// ---- 20_Product/20_ProBox/40_TC_Visualization/14_Group/V_Group.TcVIS
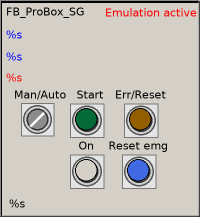
VISUALIZATION V_Group  // 200x217
VAR_IN_OUT
	{attribute 'VAR_IN_OUT_AS_POINTER'}
	fbFunction		: FB_ProBOXSG;
	fbEmuFunction	: FB_ProBOXSG_Emulation;
END_VAR
    Rectangle (0,1 200x216)
    Rectangle (6,194 177x20), "%s", text variable: fbFunction.ConfigGroup.GroupName
    Label (3,2 158x20), "FB_ProBox_SG"
    Rectangle (3,25 99x20), "%s", text variable: fbFunction.GroupData.OperationState.eState
    Rectangle (3,68 161x20), "%s", tooltip "%s", text variable: fbFunction.GroupData.ErrorData.Error.ErrorCode.Conv, invisible if: fbFunction.GroupData.ErrorData.Error.ErrorCode.Conv = 0
        p4168582468: fbFunction.GroupData.ErrorData.Error.ErrorParam
    Rectangle (3,47 99x20), "%s", text variable: fbFunction.GroupData.OperationState.eMode
    RotarySwitch (21,103 33x33), variable: fbEmuFunction.DebugManualModeSw, behaviour: TOGGLE, style: Switch-RotarySwitch-Gray
    Label (11,84 58x22), "Man/Auto"
    Rectangle (102,3 95x20), "Emulation active", invisible if: NOT ProBoxSystem.EMULATION_ENABLED
    PushSwitch (70,103 34x35), behaviour: TOGGLE, style: Switch-PushSwitch-Gray
    Ellipse (75,108 22x22), colour toggle: fbFunction.HW_Outputs.GroupStarted
        tap fbEmuFunction.DebugStartButton
    Label (71,84 38x22), "Start"
    Label (106,84 69x22), "Err/Reset"
    PushSwitch (124,103 34x35), behaviour: TOGGLE, style: Switch-PushSwitch-Gray
    Ellipse (129,108 22x22), colour toggle: fbFunction.HW_Outputs.ErrorPending
        tap fbEmuFunction.DebugResetButton
    Label (52,135 69x22), "On"
    PushSwitch (70,154 34x35), behaviour: TOGGLE, style: Switch-PushSwitch-Gray
    Ellipse (75,159 22x22), colour toggle: fbFunction.HW_Outputs.MainContactorLamp
        tap fbEmuFunction.DebugMcOnButton
    PushSwitch (122,154 34x35), behaviour: TOGGLE, style: Switch-PushSwitch-Gray
    Ellipse (127,159 22x22), colour toggle: fbFunction.HW_Outputs.EmergencyLamp
        tap fbEmuFunction.DebugResetEmgButton
    Label (104,135 69x22), "Reset emg"
END_VISUALIZATION

// ---- 20_Product/20_ProBox/40_TC_Visualization/15_PowerStore/AccessPanelCmbTxtList.TcTLO
TEXTLIST AccessPanelCmbTxtList
  1 = '1'
  2 = '2'
  3 = '3'
  4 = '4'
   = ''
END_TEXTLIST

// ---- 20_Product/20_ProBox/40_TC_Visualization/15_PowerStore/AkCmbTxtList.TcTLO
TEXTLIST AkCmbTxtList
  1 = '1'
  2 = '2'
  3 = '3'
  4 = '4'
   = ''
END_TEXTLIST

// ---- 20_Product/20_ProBox/40_TC_Visualization/15_PowerStore/LevelCmbTxtList.TcTLO
TEXTLIST LevelCmbTxtList
  1 = '1'
  2 = '2'
  3 = '3'
  4 = '4'
  5 = '5'
  6 = '6'
  7 = '7'
  8 = '8'
  9 = '9'
  10 = '10'
  11 = '11'
  12 = '12'
   = ''
END_TEXTLIST

// ---- 20_Product/20_ProBox/40_TC_Visualization/15_PowerStore/PanelCmbTxtList.TcTLO
TEXTLIST PanelCmbTxtList
  1 = '1'
  2 = '2'
  3 = '3'
  4 = '4'
   = ''
END_TEXTLIST

// ---- 20_Product/20_ProBox/40_TC_Visualization/15_PowerStore/TransferPanelCmbTxtList.TcTLO
TEXTLIST TransferPanelCmbTxtList
  1 = '1'
  2 = '2'
  3 = '3'
  4 = '4'
   = ''
END_TEXTLIST

// ---- 20_Product/20_ProBox/40_TC_Visualization/15_PowerStore/V_AccessPanel.TcVIS
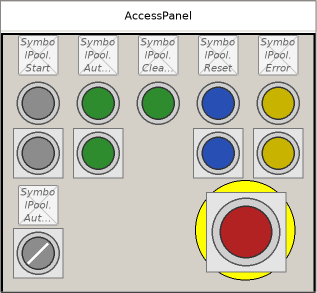
VISUALIZATION V_AccessPanel  // 317x293
VAR_IN_OUT
	Signals  : ST_AccessPanel;
END_VAR
    Rectangle (1,33 314x260)
    Image (18,35 40x40), image: SymbolPool.Start
    PushSwitch (13,128 50x50), tooltip "Activate main contactor", variable: Signals.inputs.PB_ActivateMainContactor, behaviour: TAP, style: Switch-PushSwitch-Gray
    Lamp1 (13,78 50x50), tooltip "Main contactor activated", variable: Signals.outputs.LED_MainContactorActivated, style: Lamp-Lamp1-Gray
    PushSwitch (73,128 50x50), tooltip "Auto on", variable: Signals.inputs.PB_AutoOn, behaviour: TAP, style: Switch-PushSwitch-Green
    Lamp1 (73,78 50x50), tooltip "Auto activated", variable: Signals.outputs.LED_AutoIsOn, style: Lamp-Lamp1-Green
    Lamp1 (133,78 50x50), tooltip "Clear enterance", variable: Signals.outputs.LED_ClearEnterance, style: Lamp-Lamp1-Green
    Lamp1 (193,78 50x50), tooltip "Emergency stop", variable: Signals.outputs.LED_EmergencyStop, style: Lamp-Lamp1-Blue
    PushSwitch (193,128 50x50), tooltip "Reset emergency stop", variable: Signals.inputs.PB_EmergencyStopReset, behaviour: TAP, style: Switch-PushSwitch-Blue
    Lamp1 (253,78 50x50), tooltip "Error", variable: Signals.outputs.LED_Error, style: Lamp-Lamp1-Yellow
    PushSwitch (253,128 50x50), tooltip "Reset error", variable: Signals.inputs.PB_ErrorReset, behaviour: TAP, style: Switch-PushSwitch-Yellow
    RotarySwitch (13,228 50x50), tooltip "Auto/Entry request key switch", variable: Signals.inputs.SW_EntryRequest, behaviour: TOGGLE, style: Switch-RotarySwitch-Gray
    Ellipse (195,180 100x100)
    PushSwitch (206,192 80x80), variable: Signals.inputs.PB_EmergencyStop, behaviour: TOGGLE, style: Switch-PushSwitch-Red
    Image (78,35 40x40), image: SymbolPool.AutoOn
    Image (138,35 40x40), image: SymbolPool.ClearToEnter
    Image (198,35 40x40), image: SymbolPool.Reset
    Image (258,35 40x40), image: SymbolPool.Error
    Image (18,185 40x40), image: SymbolPool.AutoMan
    Textfield (0,1 317x30), "AccessPanel"
END_VISUALIZATION

// ---- 20_Product/20_ProBox/40_TC_Visualization/15_PowerStore/V_AKcabinetPanel.TcVIS
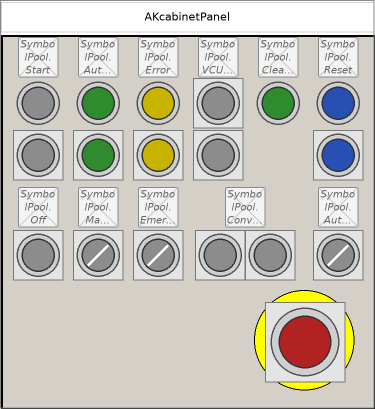
VISUALIZATION V_AKcabinetPanel  // 375x409
VAR_IN_OUT
	Signals : ST_AKcabinetPanel;
END_VAR
    Rectangle (1,35 374x374)
    Lamp1 (13,78 50x50), tooltip "Main contactor activeated", variable: Signals.outputs.LED_MainContactorActivated, style: Lamp-Lamp1-Gray
    PushSwitch (13,130 50x50), tooltip "Activate main contactor", variable: Signals.inputs.PB_ActivateMainContactor, behaviour: TAP, style: Switch-PushSwitch-Gray
    PushSwitch (73,130 50x50), tooltip "Auto on", variable: Signals.inputs.PB_AutoOn, behaviour: TAP, style: Switch-PushSwitch-Green
    Lamp1 (73,78 50x50), tooltip "Auto activated", variable: Signals.outputs.LED_AutoIsOn, style: Lamp-Lamp1-Green
    Lamp1 (133,78 50x50), tooltip "Error", variable: Signals.outputs.LED_Error, style: Lamp-Lamp1-Yellow
    PushSwitch (133,130 50x50), tooltip "Reset error", variable: Signals.inputs.PB_ErrorReset, behaviour: TAP, style: Switch-PushSwitch-Yellow
    RotarySwitch (73,230 50x50), tooltip "Man/Auto key switch", variable: Signals.inputs.SW_Auto, behaviour: TOGGLE, style: Switch-RotarySwitch-Gray
    PushSwitch (13,230 50x50), tooltip "Main contactor off", variable: Signals.inputs.PB_MainContactorOff, behaviour: TAP, style: Switch-PushSwitch-Gray
    Image (18,37 40x40), image: SymbolPool.Start
    Image (78,37 40x40), image: SymbolPool.AutoOn
    Image (138,37 40x40), image: SymbolPool.Error
    Image (18,187 40x40), image: SymbolPool.Off
    Image (78,187 40x40), image: SymbolPool.ManAuto
    Image (198,37 40x40), image: SymbolPool.VCUpDown
    PushSwitch (193,130 50x50), tooltip "VC Down", variable: Signals.inputs.PB_VcDown, behaviour: TAP, style: Switch-PushSwitch-Gray
    PushSwitch (193,78 50x50), tooltip "VC Up", variable: Signals.inputs.PB_VcUp, behaviour: TAP, style: Switch-PushSwitch-Gray
    Lamp1 (253,78 50x50), tooltip "Clear enterance", variable: Signals.outputs.LED_ClearEnterance, style: Lamp-Lamp1-Green
    Lamp1 (313,78 50x50), tooltip "Emergency stop", variable: Signals.outputs.LED_EmergencyStop, style: Lamp-Lamp1-Blue
    PushSwitch (313,130 50x50), tooltip "Reset emergency stop", variable: Signals.inputs.PB_EmergencyStopReset, behaviour: TAP, style: Switch-PushSwitch-Blue
    Image (258,37 40x40), image: SymbolPool.ClearToEnter
    Image (318,37 40x40), image: SymbolPool.Reset
    Image (225,187 40x40), image: SymbolPool.Conv_L_R
    PushSwitch (245,230 50x50), tooltip "VC Conveyor Right", variable: Signals.inputs.PB_VcConvRight, behaviour: TAP, style: Switch-PushSwitch-Gray
    PushSwitch (195,230 50x50), tooltip "VC Conveyor Left", variable: Signals.inputs.PB_VcConvLeft, behaviour: TAP, style: Switch-PushSwitch-Gray
    Image (318,187 40x40), image: SymbolPool.AutoMan
    RotarySwitch (313,230 50x50), tooltip "Auto/Entry request key switch", variable: Signals.inputs.SW_EntryRequest, behaviour: TOGGLE, style: Switch-RotarySwitch-Gray
    RotarySwitch (133,230 50x50), tooltip "Emergency drive key switch", variable: Signals.inputs.SW_EmergencyDrive, behaviour: TOGGLE, style: Switch-RotarySwitch-Gray
    Image (138,187 40x40), image: SymbolPool.EmergencyDrive
    Ellipse (254,290 100x100)
    PushSwitch (265,302 80x80), variable: Signals.inputs.PB_EmergencyStop, behaviour: TOGGLE, style: Switch-PushSwitch-Red
    Textfield (1,2 373x30), "AKcabinetPanel"
END_VISUALIZATION

// ---- 20_Product/20_ProBox/40_TC_Visualization/15_PowerStore/V_AkPanelSelecCmb.TcVIS
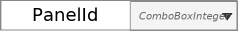
VISUALIZATION V_AkPanelSelecCmb  // 238x31
    ComboBoxInteger (130,1 108x30), variable: VisuGVL.fbPanelImp.AKPanelId, text list: 'AkCmbTxtList'
    Textfield (1,0 129x30), "PanelId"
END_VISUALIZATION

// ---- 20_Product/20_ProBox/40_TC_Visualization/15_PowerStore/V_ApSelecCmb.TcVIS
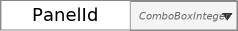
VISUALIZATION V_ApSelecCmb  // 238x31
    ComboBoxInteger (130,1 108x30), variable: VisuGVL.fbPanelImp.PanelId, text list: 'PanelCmbTxtList'
    Textfield (1,0 129x30), "PanelId"
END_VISUALIZATION

// ---- 20_Product/20_ProBox/40_TC_Visualization/15_PowerStore/V_LevelSelecCmb.TcVIS
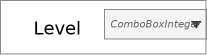
VISUALIZATION V_LevelSelecCmb  // 207x55
    ComboBoxInteger (104,9 103x30), variable: VisuGVL.fbPanelImp.Level, text list: 'LevelCmbTxtList'
    Label (5,2 105x53), "Level"
END_VISUALIZATION

// ---- 20_Product/20_ProBox/40_TC_Visualization/15_PowerStore/V_PanelSelecCmb.TcVIS
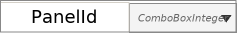
VISUALIZATION V_PanelSelecCmb  // 237x33
    ComboBoxInteger (129,3 108x30), variable: VisuGVL.fbPanelImp.PanelId, text list: 'PanelCmbTxtList'
    Textfield (0,2 129x30), "PanelId"
END_VISUALIZATION

// ---- 20_Product/20_ProBox/40_TC_Visualization/15_PowerStore/V_TpSelecCmb.TcVIS
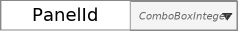
VISUALIZATION V_TpSelecCmb  // 238x31
    ComboBoxInteger (130,1 108x30), variable: VisuGVL.fbPanelImp.PanelId, text list: 'PanelCmbTxtList'
    Textfield (1,0 129x30), "PanelId"
END_VISUALIZATION

// ---- 20_Product/20_ProBox/40_TC_Visualization/15_PowerStore/V_TransferPanel.TcVIS
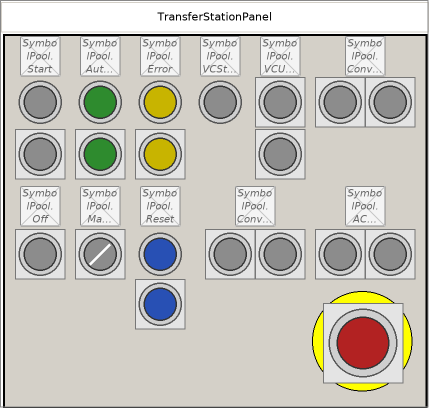
VISUALIZATION V_TransferPanel  // 429x408
VAR_IN_OUT
	Signals : ST_TransferPanel;
END_VAR
    Rectangle (3,34 424x374)
    Ellipse (312,291 100x100)
    PushSwitch (15,129 50x50), tooltip "Activate main contactor", variable: Signals.inputs.PB_ActivateMainContactor, behaviour: TAP, style: Switch-PushSwitch-Gray
    Lamp1 (15,77 50x50), tooltip "Main contactor activeated", variable: Signals.outputs.LED_MainContactorActivated, style: Lamp-Lamp1-Gray
    PushSwitch (75,129 50x50), tooltip "Auto on", variable: Signals.inputs.PB_AutoOn, behaviour: TAP, style: Switch-PushSwitch-Green
    Lamp1 (75,77 50x50), tooltip "Auto activated", variable: Signals.outputs.LED_AutoIsOn, style: Lamp-Lamp1-Green
    Lamp1 (135,77 50x50), tooltip "Error", variable: Signals.outputs.LED_Error, style: Lamp-Lamp1-Yellow
    PushSwitch (135,129 50x50), tooltip "Reset error", variable: Signals.inputs.PB_ErrorReset, behaviour: TAP, style: Switch-PushSwitch-Yellow
    Lamp1 (135,229 50x50), tooltip "Emergency stop", variable: Signals.outputs.LED_EmergencyStop, style: Lamp-Lamp1-Blue
    PushSwitch (135,279 50x50), tooltip "Reset emergency stop", variable: Signals.inputs.PB_EmergencyStopReset, behaviour: TAP, style: Switch-PushSwitch-Blue
    RotarySwitch (75,229 50x50), tooltip "Man/Auto", variable: Signals.inputs.SW_Auto, behaviour: TOGGLE, style: Switch-RotarySwitch-Gray
    Lamp1 (195,77 50x50), tooltip "VC stopped", variable: Signals.outputs.LED_VcStopped, style: Lamp-Lamp1-Gray
    PushSwitch (255,129 50x50), tooltip "VC Down", variable: Signals.inputs.PB_VcDown, behaviour: TAP, style: Switch-PushSwitch-Gray
    PushSwitch (255,77 50x50), tooltip "VC Up", variable: Signals.inputs.PB_VcUp, behaviour: TAP, style: Switch-PushSwitch-Gray
    PushSwitch (365,77 50x50), tooltip "Transfer Conveyor Right", variable: Signals.inputs.PB_Conv_1_Right, behaviour: TAP, style: Switch-PushSwitch-Gray
    PushSwitch (315,77 50x50), tooltip "Transfer Conveyor Left", variable: Signals.inputs.PB_Conv_1_Left, behaviour: TAP, style: Switch-PushSwitch-Gray
    PushSwitch (255,229 50x50), tooltip "VC Conveyor Right", variable: Signals.inputs.PB_VcConvRight, behaviour: TAP, style: Switch-PushSwitch-Gray
    PushSwitch (205,229 50x50), tooltip "VC Conveyor Left", variable: Signals.inputs.PB_VcConvLeft, behaviour: TAP, style: Switch-PushSwitch-Gray
    PushSwitch (365,229 50x50), tooltip "AC Conveyor Right", variable: Signals.inputs.PB_AC_ConvRight, behaviour: TAP, style: Switch-PushSwitch-Gray
    PushSwitch (315,229 50x50), tooltip "AC Conveyor Left", variable: Signals.inputs.PB_AC_ConvLeft, behaviour: TAP, style: Switch-PushSwitch-Gray
    PushSwitch (15,229 50x50), tooltip "Main contactor off", variable: Signals.inputs.PB_MainContactorOff, behaviour: TAP, style: Switch-PushSwitch-Gray
    PushSwitch (323,303 80x80), tooltip "Emergency stop", variable: Signals.inputs.PB_EmergencyStop, behaviour: TOGGLE, style: Switch-PushSwitch-Red
    Image (20,36 40x40), image: SymbolPool.Start
    Image (80,36 40x40), image: SymbolPool.AutoOn
    Image (140,36 40x40), image: SymbolPool.Error
    Image (200,36 40x40), image: SymbolPool.VCStopped
    Image (260,36 40x40), image: SymbolPool.VCUpDown
    Image (345,36 40x40), image: SymbolPool.Conv1_L_R
    Image (235,186 40x40), image: SymbolPool.Conv_L_R
    Image (345,186 40x40), image: SymbolPool.AC_Conv_L_R
    Image (20,186 40x40), image: SymbolPool.Off
    Image (80,186 40x40), image: SymbolPool.ManAuto
    Image (140,186 40x40), image: SymbolPool.Reset
    Textfield (1,2 428x30), "TransferStationPanel"
END_VISUALIZATION

// ---- 20_Product/20_ProBox/40_TC_Visualization/15_PowerStore/V_VC_AccessPanel.TcVIS
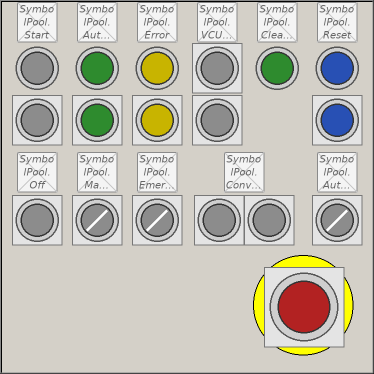
VISUALIZATION V_VC_AccessPanel  // 374x374
VAR_IN_OUT
	Signals : ST_VC_AccessPanel;
END_VAR
    Rectangle (0,0 374x374)
    Lamp1 (12,43 50x50), tooltip "Main contactor activeated", variable: Signals.outputs.LED_MainContactorActivated, style: Lamp-Lamp1-Gray
    PushSwitch (12,95 50x50), tooltip "Activate main contactor", variable: Signals.inputs.PB_ActivateMainContactor, behaviour: TAP, style: Switch-PushSwitch-Gray
    PushSwitch (72,95 50x50), tooltip "Auto on", variable: Signals.inputs.PB_AutoOn, behaviour: TAP, style: Switch-PushSwitch-Green
    Lamp1 (72,43 50x50), tooltip "Auto activated", variable: Signals.outputs.LED_AutoIsOn, style: Lamp-Lamp1-Green
    Lamp1 (132,43 50x50), tooltip "Error", variable: Signals.outputs.LED_Error, style: Lamp-Lamp1-Yellow
    PushSwitch (132,95 50x50), tooltip "Reset error", variable: Signals.inputs.PB_ErrorReset, behaviour: TAP, style: Switch-PushSwitch-Yellow
    RotarySwitch (72,195 50x50), tooltip "Man/Auto key switch", variable: Signals.inputs.SW_Auto, behaviour: TOGGLE, style: Switch-RotarySwitch-Gray
    PushSwitch (12,195 50x50), tooltip "Main contactor off", variable: Signals.inputs.PB_MainContactorOff, behaviour: TAP, style: Switch-PushSwitch-Gray
    Image (17,2 40x40), image: SymbolPool.Start
    Image (77,2 40x40), image: SymbolPool.AutoOn
    Image (137,2 40x40), image: SymbolPool.Error
    Image (17,152 40x40), image: SymbolPool.Off
    Image (77,152 40x40), image: SymbolPool.ManAuto
    Image (197,2 40x40), image: SymbolPool.VCUpDown
    PushSwitch (192,95 50x50), tooltip "VC Down", variable: Signals.inputs.PB_VcDown, behaviour: TAP, style: Switch-PushSwitch-Gray
    PushSwitch (192,43 50x50), tooltip "VC Up", variable: Signals.inputs.PB_VcUp, behaviour: TAP, style: Switch-PushSwitch-Gray
    Lamp1 (252,43 50x50), tooltip "Clear enterance", variable: Signals.outputs.LED_ClearEnterance, style: Lamp-Lamp1-Green
    Lamp1 (312,43 50x50), tooltip "Emergency stop", variable: Signals.outputs.LED_EmergencyStop, style: Lamp-Lamp1-Blue
    PushSwitch (312,95 50x50), tooltip "Reset emergency stop", variable: Signals.inputs.PB_EmergencyStopReset, behaviour: TAP, style: Switch-PushSwitch-Blue
    Image (257,2 40x40), image: SymbolPool.ClearToEnter
    Image (317,2 40x40), image: SymbolPool.Reset
    Image (224,152 40x40), image: SymbolPool.Conv_L_R
    PushSwitch (244,195 50x50), tooltip "VC Conveyor Right", variable: Signals.inputs.PB_VcConvRight, behaviour: TAP, style: Switch-PushSwitch-Gray
    PushSwitch (194,195 50x50), tooltip "VC Conveyor Left", variable: Signals.inputs.PB_VcConvLeft, behaviour: TAP, style: Switch-PushSwitch-Gray
    Image (317,152 40x40), image: SymbolPool.AutoMan
    RotarySwitch (312,195 50x50), tooltip "Auto/Entry request key switch", variable: Signals.inputs.SW_EntryRequest, behaviour: TOGGLE, style: Switch-RotarySwitch-Gray
    RotarySwitch (132,195 50x50), tooltip "Emergency drive key switch", variable: Signals.inputs.SW_EmergencyDrive, behaviour: TOGGLE, style: Switch-RotarySwitch-Gray
    Image (137,152 40x40), image: SymbolPool.EmergencyDrive
    Ellipse (253,255 100x100)
    PushSwitch (264,267 80x80), variable: Signals.inputs.PB_EmergencyStop, behaviour: TOGGLE, style: Switch-PushSwitch-Red
END_VISUALIZATION

// ---- 20_Product/20_ProBox/40_TC_Visualization/99_SIS/V_SIS_Control.TcVIS
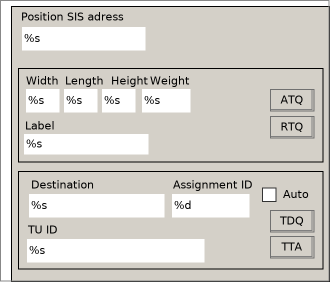
VISUALIZATION V_SIS_Control  // 330x282
VAR_IN_OUT	
	{attribute 'VAR_IN_OUT_AS_POINTER'}
	fb_VizuSIS	: FB_VizuSIS;	
		
END_VAR
    Rectangle (11,6 319x276)
    Textfield (21,26 125x25), "%s", text variable: fb_VizuSIS.PositionString, colour toggle: fb_VizuSIS.BadPosition
        OnMouseClick: write the text variable via Edit
    Label (18,7 117x20), "Position SIS adress"
    Rectangle (18,68 305x94)
    Button (270,89 44x22), "ATQ"
        tap fb_VizuSIS.ATQ
    Textfield (25,88 35x25), "%s", text variable: fb_VizuSIS.ATQ_Dimension.Width
        OnMouseClick: write the text variable via Edit
    Textfield (101,88 35x25), "%s", text variable: fb_VizuSIS.ATQ_Dimension.Height
        OnMouseClick: write the text variable via Edit
    Textfield (63,88 35x25), "%s", text variable: fb_VizuSIS.ATQ_Dimension.Length
        OnMouseClick: write the text variable via Edit
    Textfield (141,88 50x25), "%s", text variable: fb_VizuSIS.ATQ_Dimension.Weight
        OnMouseClick: write the text variable via Edit
    Label (23,71 41x20), "Width"
    Label (62,71 48x20), "Length"
    Label (108,71 41x20), "Height"
    Label (147,71 48x20), "Weight"
    Textfield (23,133 126x22), "%s", text variable: fb_VizuSIS.ATQ_Label
        OnMouseClick: write the text variable via Edit
    Button (270,116 44x22), "RTQ"
        tap fb_VizuSIS.RTQ
    Rectangle (18,171 305x98)
    Button (270,236 44x22), "TTA"
        tap fb_VizuSIS.TTA
    Textfield (28,193 137x25), "%s", text variable: fb_VizuSIS.TTA_Destination
        OnMouseClick: write the text variable via Edit
    Button (270,210 44x22), "TDQ"
        tap fb_VizuSIS.TDQ
    Label (25,220 117x20), "TU ID"
    Textfield (26,238 179x25), "%s", text variable: fb_VizuSIS.TU_ID, input disabled if: fb_VizuSIS.AutoID
        OnMouseClick: write the text variable via Edit, min 18, max 18
    Label (28,175 117x20), "Destination"
    Label (22,116 117x20), "Label"
    Textfield (171,193 79x25), "%d", text variable: fb_VizuSIS.AssignmentID, input disabled if: fb_VizuSIS.AutoID
        OnMouseClick: write the text variable via Edit
    Label (170,175 90x20), "Assignment ID"
    Checkbox (260,183 51x23), "Auto", tooltip "Reuse TU ID and Assignment ID from TU Table", variable: fb_VizuSIS.AutoID
END_VISUALIZATION

// ---- 20_Product/20_ProBox/ProBox_Version.TcTLO
TEXTLIST ProBox_Version
  Version = 'R1.13.0'
  Company = 'Swisslog/PTC'
   = ''
END_TEXTLIST
